(* CODESYS project Cat2.project

Project tree, tasks and I/O mapping:
  Device : CODESYS Control RTE V3, 3S - Smart Software Solutions GmbH, order no. 305017, version 3.5.11.0
    application Application
      libraries: Standard, * (System)
      task MainTask (cyclic, interval t#20ms, priority 1) calls PLC_PRG
      task VISU_TASK (cyclic, interval 100 ms, priority 31) calls VisuElems.Visu_Prg
      program PLC_PRG [ST]
      visualisation Visualization
      function block FB_Plant [ST]
      function block FB_Controller [ST]
      global variables GVL
      data type ST_PlantToController
      data type ST_ControllerToPlant
  text list GlobalTextList
  GlobalImagePool
*)

// Device/Application/ST_PlantToController
TYPE ST_PlantToController :
STRUCT
	// Buttons
	bCalibration : BOOL;
	bClean : BOOL;
	
	// Door
	bDoorOpened : BOOL;
	bDoorClosed : BOOL;
	
	// Separator
	bSeparatorUp : BOOL;
	bSeparatorDown : BOOL;
	
	// Weight
	CurrentWeight : REAL;
	
	// Wastes
	CurrentWastes : REAL;
	
	// Aroma
	CurrentAroma : REAL;

END_STRUCT
END_TYPE

// Device/Application/ST_ControllerToPlant
TYPE ST_ControllerToPlant :
STRUCT
	// Calibration
	bCalibration : BOOL;

	// Door
	bOpenDoor : BOOL;
	bCloseDoor : BOOL;
	bDoorStop : BOOL;
	
	// Separator
	bSeparatorUp : BOOL;
	bSeparatorDown : BOOL;
	
	// Aroma
	bAromaOn : BOOL;
	DeleteAroma : BOOL;
	
	// Wastes
	AddWastes : BOOL;
	
	// Weight
	FillerWeight : REAL;
	DeleteFiller : BOOL;
	
	bLowFiller : BOOL;
	bCriticalWastes : BOOL;
	bLowAroma : BOOL;
	AromaWorking : BOOL;
	
	UVworking : BOOL;
	
END_STRUCT
END_TYPE

// Device/Application/GVL

VAR_GLOBAL
	// Messages
	PlantToController : ST_PlantToController;
	ControllerToPlant : ST_ControllerToPlant;
	
	// Buttons
	CalibrationBtn : BOOL;
	CleanBtn : BOOL;
	
	AddCatBtn : BOOL;
	RemoveCatBtn : BOOL;
	
	RemoveWastesBtn : BOOL;
	RefillAromaBtn : BOOL;
	
	// Movements
	SeparatorPosition : REAL := 0.0;
	DoorPosition : REAL := 0.0;
	CatState : BOOL := FALSE;
	
	// Leds
	CalibrationLed : BOOL := FALSE;
	UVLed : BOOL;
	LowFillerLed : BOOL;
	FullWastesLed : BOOL;
	LowAromaLed : BOOL;
	AromaLed : BOOL;
	
	AddedFiller : REAL;
	CatWeight : REAL := 3.5;

END_VAR

// Device/Application/PLC_PRG
PROGRAM PLC_PRG
VAR
	Plant : FB_Plant;
	Controller : FB_Controller;
END_VAR

Plant();
Controller();

END_PROGRAM

// Device/Application/FB_Plant
FUNCTION_BLOCK FB_Plant
VAR_INPUT
END_VAR
VAR_OUTPUT
END_VAR

VAR CONSTANT
	FillerPart : REAL := 0.2;
	WastesPart : REAL := 5.0;
	AromaPart : REAL := 0.2;
	
	DoorMin : REAL := 0.0;
	DoorMax : REAL := 100.0;
	
	SeparatorMin : REAL := 270.0;
	SeparatorMax : REAL := 360.0;
END_VAR

VAR
	// Controller flags
	IsCalibration : BOOL := FALSE;
	IsCat : BOOL := FALSE;

	// Button triggers
	rtCalib : R_TRIG;
	CalibEvent : BOOL := FALSE;
	
	rtClean : R_TRIG;
	CleanEvent : BOOL := FALSE;
	
	rtAddCat : R_TRIG;
	rtRemoveCat : R_TRIG;
	
	rtRemoveWastes : R_TRIG;
	rtRefillAroma : R_TRIG;
	
	
	// Door movement
	DoorClose : BOOL := FALSE;
	DoorOpen : BOOL := FALSE;
	DoorOpening : BOOL := FALSE;
	DoorClosing : BOOL := FALSE;
	DoorClosed : BOOL := FALSE;
	DoorOpened : BOOL := FALSE;
	DoorPosition : REAL := DoorMin;
	
	// Separator movement
	SeparatorUp : BOOL := FALSE;
	flSepUp : F_TRIG;
	SeparatorDown : BOOL := FALSE;
	SeparatorUpping : BOOL := FALSE;
	SeparatorDowning : BOOL := FALSE;
	SeparatorUpped : BOOL := FALSE;
	SeparatorDowned : BOOL := FALSE;
	SeparatorPosition : REAL := SeparatorMax;
	
	// Weight
	CurrentWeight : REAL := 0.0;
	FillerWeight : REAL := 0.0;
	DeleteFiller : BOOL := FALSE;
	LowFiller : BOOL := FALSE;
	
	// Wastes
	CurrentWastesLevel : REAL := 0.0;
	AddWastes : BOOL := FALSE;
	CriticalWastes : BOOL := FALSE;
	
	// Aroma
	CurrentAromaLevel : REAL := 100.0;
	DeleteAroma : BOOL := FALSE;
	LowAroma : BOOL := FALSE;
	AromaWorking : BOOL := FALSE;
	flAroma : F_TRIG;
	
	UVworking : BOOL := FALSE;

END_VAR

// ==================== From Controller =======================
IsCalibration := GVL.ControllerToPlant.bCalibration;

DoorClose := GVL.ControllerToPlant.bCloseDoor;
DoorOpen := GVL.ControllerToPlant.bOpenDoor;
SeparatorUp := GVL.ControllerToPlant.bSeparatorUp;
SeparatorDown := GVL.ControllerToPlant.bSeparatorDown;

FillerWeight := GVL.ControllerToPlant.FillerWeight;
DeleteFiller := GVL.ControllerToPlant.DeleteFiller;

AddWastes := GVL.ControllerToPlant.AddWastes;

DeleteAroma := GVL.ControllerToPlant.DeleteAroma;

LowFiller := GVL.ControllerToPlant.bLowFiller;
LowAroma := GVL.ControllerToPlant.bLowAroma;
CriticalWastes := GVL.ControllerToPlant.bCriticalWastes;

UVworking := GVL.ControllerToPlant.UVworking;
AromaWorking := GVL.ControllerToPlant.AromaWorking;

// ==================== Button Events =======================
rtCalib(CLK := GVL.CalibrationBtn);
CalibEvent := rtCalib.Q;

rtAddCat(CLK := GVL.AddCatBtn);
rtRemoveCat(CLK := GVL.RemoveCatBtn);
IF rtAddCat.Q AND DoorOpened AND NOT IsCalibration THEN
	IsCat := TRUE;
ELSIF rtRemoveCat.Q AND DoorOpened THEN
	IsCat := FALSE;
END_IF

rtClean(CLK := GVL.CleanBtn);
CleanEvent := rtClean.Q;

rtRemoveWastes(CLK := GVL.RemoveWastesBtn);
rtRefillAroma(CLK := GVL.RefillAromaBtn);

IF rtRemoveWastes.Q AND NOT (SeparatorUpping OR SeparatorDowning) THEN
	CurrentWastesLevel := 0.0;
END_IF

IF rtRefillAroma.Q AND NOT AromaWorking THEN
	CurrentAromaLevel := 100.0;
END_IF

// ==================== Main =======================

// Calibration
IF IsCalibration THEN
	CurrentWeight := GVL.AddedFiller;
ELSIF IsCat THEN
	CurrentWeight := FillerWeight + GVL.CatWeight;
ELSE
	CurrentWeight := FillerWeight;
END_IF

// Door moving
IF DoorClose THEN
	DoorClosing := TRUE;
	DoorOpening := FALSE;
END_IF
	
IF DoorOpen THEN
	DoorClosing := FALSE;
	DoorOpening := TRUE;
END_IF

IF DoorOpen AND DoorClose THEN
	DoorClosing := FALSE;
	DoorOpening := FALSE;
END_IF

IF DoorClosing AND DoorPosition < DoorMax THEN
	DoorPosition := DoorPosition + 1;
	DoorClosed := FALSE;
	DoorOpened := FALSE;
ELSIF DoorOpening AND DoorPosition > DoorMin THEN
	DoorPosition := DoorPosition - 1;
	DoorClosed := FALSE;
	DoorOpened := FALSE;
END_IF

IF DoorPosition >= DoorMax THEN
	DoorPosition := DoorMax;
	DoorClosed := TRUE;
	DoorOpened := FALSE;
ELSIF DoorPosition <= DoorMin THEN
	DoorPosition := DoorMin;
	DoorOpened := TRUE;
	DoorClosed := FALSE;
END_IF

// Separator moving
flSepUp(CLK := SeparatorUp);

IF flSepUp.Q THEN
	IF (100 - CurrentWastesLevel) >= WastesPart THEN
		CurrentWastesLevel := CurrentWastesLevel + WastesPart;
	END_IF
	
	IF FillerWeight >= FillerPart THEN
		FillerWeight := FillerWeight - FillerPart;
		CurrentWeight := FillerWeight;
	END_IF
END_IF

IF SeparatorUp THEN
	SeparatorUpping := TRUE;
	SeparatorDowning := FALSE;
END_IF

IF SeparatorDown THEN
	SeparatorUpping := FALSE;
	SeparatorDowning := TRUE;
END_IF

IF SeparatorUp AND SeparatorDown THEN
	SeparatorUpping := FALSE;
	SeparatorDowning := FALSE;
END_IF

IF SeparatorUpping AND SeparatorPosition > SeparatorMin THEN
	SeparatorPosition := SeparatorPosition - 1;
	SeparatorUpped := FALSE;
	SeparatorDowned := FALSE;
ELSE
	SeparatorUpping := FALSE;
END_IF

IF SeparatorDowning AND SeparatorPosition < SeparatorMax THEN
	SeparatorPosition := SeparatorPosition + 1;
	SeparatorUpped := FALSE;
	SeparatorDowned := FALSE;
ELSE
	SeparatorDowning := FALSE;
END_IF

IF SeparatorPosition <= SeparatorMin THEN
	SeparatorPosition := SeparatorMin;
	SeparatorUpped := TRUE;
	SeparatorDowned := FALSE;
ELSIF SeparatorPosition >= SeparatorMax THEN
	SeparatorPosition := SeparatorMax;
	SeparatorUpped := FALSE;
	SeparatorDowned := TRUE;
END_IF

flAroma(CLK := AromaWorking);
IF flAroma.Q THEN
	IF CurrentAromaLevel >= AromaPart THEN
		CurrentAromaLevel := CurrentAromaLevel - AromaPart;
	END_IF
END_IF

// ==================== Positions =======================
GVL.DoorPosition := DoorPosition;
GVL.SeparatorPosition := SeparatorPosition;

// ==================== Leds =======================
GVL.CalibrationLed := IsCalibration;

GVL.CatState := IsCat;

GVL.FullWastesLed := CriticalWastes;
GVL.LowFillerLed := LowFiller;
GVL.LowAromaLed := LowAroma;

GVL.UVLed := UVworking;
GVL.AromaLed := AromaWorking;

// ==================== To Controller =======================
GVL.PlantToController.bCalibration := CalibEvent;
GVL.PlantToController.bClean := CleanEvent;

GVL.PlantToController.bDoorClosed := DoorClosed;
GVL.PlantToController.bDoorOpened := DoorOpened;
GVL.PlantToController.bSeparatorUp := SeparatorUpped;
GVL.PlantToController.bSeparatorDown := SeparatorDowned;

GVL.PlantToController.CurrentWeight := CurrentWeight;

GVL.PlantToController.CurrentWastes := CurrentWastesLevel;

GVL.PlantToController.CurrentAroma := CurrentAromaLevel;

END_FUNCTION_BLOCK

// Device/Application/FB_Controller
FUNCTION_BLOCK FB_Controller
VAR_INPUT
END_VAR
VAR_OUTPUT
END_VAR

VAR CONSTANT
	// Delay
	CatDelay : TIME := T#3S;
	SeparatorDelay : TIME := T#1S;
	UVdelay : TIME := T#4S;
	AromaDelay : TIME := T#2S;
	
	// Weight
	WeightTolerance : REAL := 0.02;
	LowFillerLevel : REAL := 0.5;
	LowAromaLevel : REAL := 0.05;
	CriticalWastesLevel : REAL := 90.0;
	
	VisitsToClean : INT := 5;
	
END_VAR

VAR
	LastState : INT := 0;
	CleaningState : INT := 0;
	State : INT := 0;
	
	VisitsCount : INT := 0;
	
	// Events
	CalibEvent : BOOL := FALSE;
	CleanEvent : BOOL := FALSE;
	
	// Flags
	CalibNow : BOOL := FALSE;
	
	CatNow : BOOL := FALSE;
	CatLeaved : BOOL := FALSE;
	CatDelayTimer : TON;
	
	CleaningNow : BOOL := FALSE;
	DoorMovingNow : BOOL := FALSE;
	
	UVnow : BOOL := FALSE;
	UVtimer : TON;
	
	AromaNow : BOOL := FALSE;
	
	// Door
	DoorClosed : BOOL := FALSE;
	DoorOpened : BOOL := FALSE;
	DoorOpening : BOOL := FALSE;
	DoorClosing : BOOL := FALSE;
	
	// Separator
	SeparatorUp : BOOL := FALSE;
	SeparatorDown : BOOL := FALSE;
	SeparatorUpping : BOOL := FALSE;
	SeparatorDowning : BOOL := FALSE;
	SeparatorDelayTimer : TON;
	SeparatorInDelay : BOOL := FALSE;
	
	// Weight
	CurrentWeight : REAL := 0;
	FillerWeight : REAL := 0;
	LowFiller : BOOL := FALSE;
	DeleteFiller : BOOL := FALSE;
	
	// Aroma
	CurrentAroma : REAL := 100.0;
	DeleteAroma : BOOL := FALSE;
	AromaTimer : TON;
	CriticalAroma : BOOL := FALSE;
	
	// Wastes
	CurrentWastes : REAL := 0.0;
	AddWastes : BOOL := FALSE;
	CriticalWastes : BOOL := FALSE;
	
END_VAR

CalibEvent := GVL.PlantToController.bCalibration;
CleanEvent := GVL.PlantToController.bClean;

DoorClosed := GVL.PlantToController.bDoorClosed;
DoorOpened := GVL.PlantToController.bDoorOpened;
SeparatorUp := GVL.PlantToController.bSeparatorUp;
SeparatorDown := GVL.PlantToController.bSeparatorDown;

CurrentWeight := GVL.PlantToController.CurrentWeight;
CurrentAroma := GVL.PlantToController.CurrentAroma;
CurrentWastes := GVL.PlantToController.CurrentWastes;

// Timers
CatDelayTimer(IN := CatLeaved, PT := SeparatorDelay);
SeparatorDelayTimer(IN := SeparatorInDelay, PT := SeparatorDelay);
UVtimer(IN := UVnow, PT := AromaDelay);
AromaTimer(IN := AromaNow, PT := AromaDelay);

DeleteFiller := FALSE;
AddWastes := FALSE;
DeleteAroma := FALSE;

IF DoorClosed AND State <> 1 THEN
	FillerWeight := CurrentWeight;
END_IF


CASE State OF
	0: // Zero state
		// Calibration event
		IF CalibEvent THEN
			LastState := 0;
			State := 10;
			RETURN;
		END_IF
		
		// Low aroma level
		IF CurrentAroma <= LowAromaLevel THEN
			CriticalAroma := TRUE;
		ELSE
			CriticalAroma := FALSE;
		END_IF
		
		// Critical wastes
		IF CurrentWastes >= CriticalWastesLevel THEN
			CriticalWastes := TRUE;
			State := 2;
			RETURN;
		ELSE
			CriticalWastes := FALSE;
		END_IF
		
		// Low filler
		IF FillerWeight <= LowFillerLevel THEN 
			LowFiller := TRUE;
			State := 1;
			RETURN;
		ELSE
			LowFiller := FALSE;
		END_IF
		
		// Cat in the litter box
		IF ABS(CurrentWeight - FillerWeight) > WeightTolerance THEN
			LastState := 0;
			State := 20;
			RETURN;
		ELSE
			FillerWeight := CurrentWeight;
		END_IF
		
		// Clean
		IF CleanEvent THEN
			LastState := 0;
			State := 40;
			RETURN;
		END_IF
		
	1: // Low filler level
		IF CalibEvent THEN
			State := 10;
		END_IF
		
	2: // Full wastes box
		IF CurrentWastes < CriticalWastesLevel THEN
			CriticalWastes := FALSE;
			State := 0;
		END_IF
		
	10: // Calibration
		CalibNow := TRUE;
		FillerWeight := CurrentWeight;
		IF CalibEvent THEN
			CalibNow := FALSE;
			State := 0;
		END_IF;
		
	20: // Cat here
		IF ABS(CurrentWeight - FillerWeight) <= WeightTolerance THEN
			CatLeaved := TRUE;
			VisitsCount := VisitsCount + 1;
			State := State + 1;
		END_IF
	
	21:
		IF ABS(CurrentWeight - FillerWeight) > WeightTolerance THEN
			CatLeaved := FALSE;
			State := State - 1;
		ELSIF CatDelayTimer.Q THEN
			CatLeaved := FALSE;
			State := State + 1;
		END_IF
	
	22:
		LastState := 22;
		State := 30;
		
	30: // Clening loop
		CASE LastState OF
			22: // Closing door
				State := 90;
			90: // Upping separator
				State := 100;
			100:
				SeparatorInDelay := TRUE;
				State := 102;
			102: // Downing separator
				SeparatorInDelay := FALSE;
				State := 101;
			101: // Opening door
				DeleteFiller := TRUE;
				AddWastes := TRUE;
				IF VisitsCount >= VisitsToClean THEN
					State := 40;
				ELSE
					State := 91;
				END_IF
			40:
				State := 91;
			91: // Finish
				State := 0;
				
		END_CASE
		LastState := 30;
	
	40: // UV and aroma
		CASE LastState OF
			0:
				CleaningState := 0;
				State := 90;
			30:
				UVnow := TRUE;
				CleaningState := 30;
				State := 110;
			90:
				UVnow := TRUE;
				State := 110;
			91:
				State := 0;
			110:
				UVnow := FALSE;
				AromaNow := NOT CriticalAroma;
				State := 120;
			120:
				VisitsCount := 0;
				AromaNow := FALSE;
				DeleteAroma := TRUE;
				IF CleaningState = 0 THEN
					State := 91;
				ELSE
					State := CleaningState;	
				END_IF			
		END_CASE
		LastState := 40;
		
	90: // Closing door
		DoorClosing := TRUE;
		IF DoorClosed THEN
			DoorClosing := FALSE;
			State := LastState;
			LastState := 90;
		END_IF
	
	91: // Opening door
		DoorOpening := TRUE;
		IF DoorOpened THEN
			DoorOpening := FALSE;
			State := LastState;
			LastState := 91;
		END_IF
		
	100: // Separator upping
		SeparatorUpping := TRUE;
		IF SeparatorUp THEN
			SeparatorUpping := FALSE;
			State := LastState;
			LastState := 100;
		END_IF
		
	101: // Separator downing
		SeparatorDowning := TRUE;
		IF SeparatorDown THEN
			SeparatorDowning := FALSE;
			State := LastState;
			LastState := 101;
		END_IF
	
	102: // Separator weiting
		IF SeparatorDelayTimer.Q THEN
			State := LastState;
			LastState := 102;
		END_IF
		
	110: // UV Cleaning
		IF UVtimer.Q THEN
			State := LastState;
			LastState := 110;
		END_IF
		
	120: // Aroma Working
		IF AromaTImer.Q OR CriticalAroma THEN
			State := LastState;
			LastState := 120;
		END_IF
END_CASE

GVL.ControllerToPlant.bCalibration := CalibNow;

GVL.ControllerToPlant.bCloseDoor := DoorClosing;
GVL.ControllerToPlant.bOpenDoor := DoorOpening;
GVL.ControllerToPlant.bSeparatorUp := SeparatorUpping;
GVL.ControllerToPlant.bSeparatorDown := SeparatorDowning;

GVL.ControllerToPlant.UVworking := UVnow;
GVL.ControllerToPlant.AromaWorking := AromaNow;

GVL.ControllerToPlant.FillerWeight := FillerWeight;
GVL.ControllerToPlant.DeleteFiller := DeleteFiller;

GVL.ControllerToPlant.AddWastes := AddWastes;
GVL.ControllerToPlant.DeleteAroma := DeleteAroma;

GVL.ControllerToPlant.bLowAroma := CriticalAroma;
GVL.ControllerToPlant.bLowFiller := LowFiller;
GVL.ControllerToPlant.bCriticalWastes := CriticalWastes;

END_FUNCTION_BLOCK

// Device/Application/Visualization
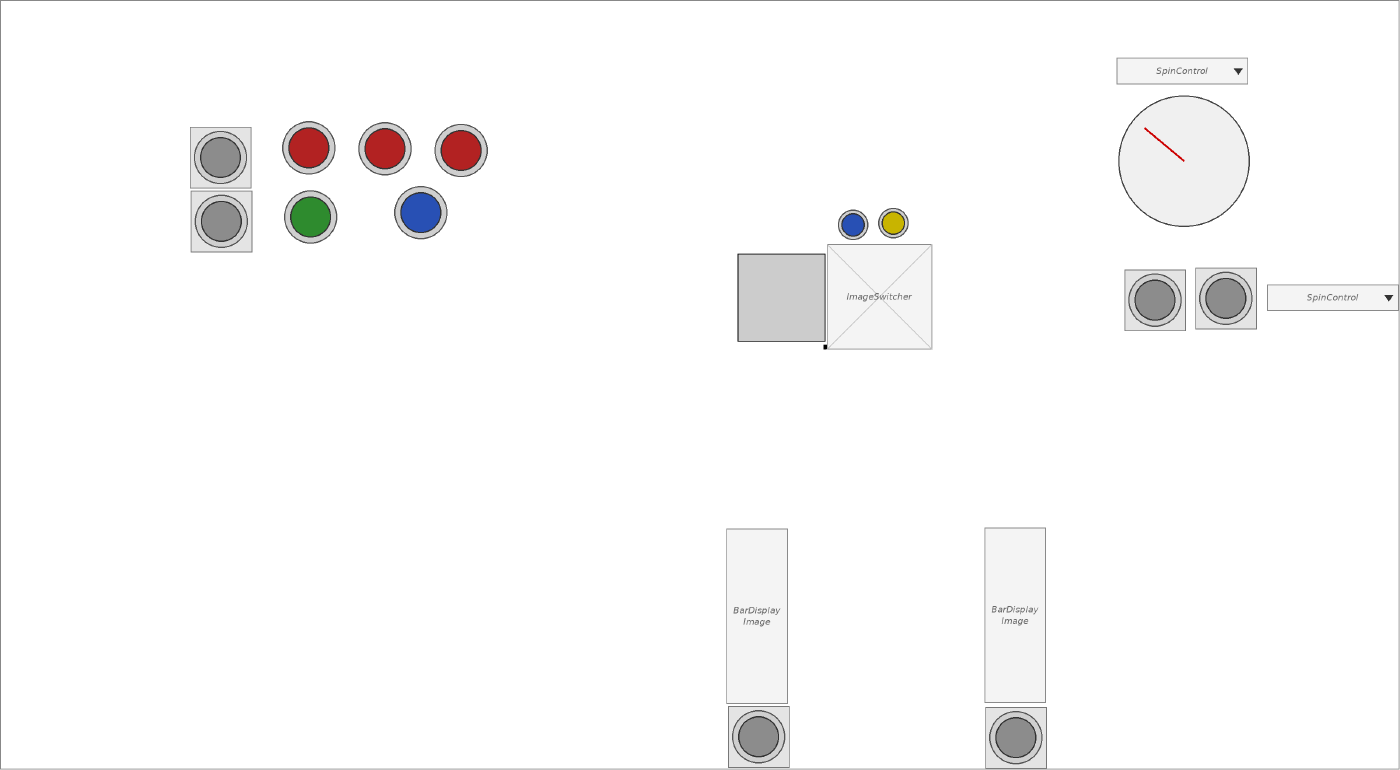
VISUALIZATION Visualization  // 1600x880
    PushSwitch (217,145 70x70), variable: CleanBtn, behaviour: TOGGLE, style: Switch-PushSwitch-Gray
    Rectangle (941,394 100x5)
        p2858320360: SeparatorPosition
    RoundedRectangle (843,290 100x100)
        p3560616238: DoorPosition
    ImageSwitcher (945,279 120x120), variable: CatState, background image: cat, behaviour: TOGGLE
    PushSwitch (218,218 70x70), variable: CalibrationBtn, behaviour: TOGGLE, style: Switch-PushSwitch-Gray
    PushSwitch (1285,308 70x70), variable: RemoveCatBtn, behaviour: TOGGLE, style: Switch-PushSwitch-Gray
    PushSwitch (1366,306 70x70), variable: AddCatBtn, behaviour: TOGGLE, style: Switch-PushSwitch-Gray
    PushSwitch (1126,808 70x70), variable: RefillAromaBtn, behaviour: TOGGLE, style: Switch-PushSwitch-Gray
    PushSwitch (832,807 70x70), variable: RemoveWastesBtn, behaviour: TOGGLE, style: Switch-PushSwitch-Gray
    BarDisplayImage (1125,603 70x200), value: PlantToController.CurrentAroma, style: BarDisplayImage-Gray, scale format: %.1f, scale 0..100
    BarDisplayImage (830,604 70x200), value: PlantToController.CurrentWastes, style: BarDisplayImage-Gray, scale format: %.1f, scale 0..100
    SpinControl (1448,325 150x30), variable: CatWeight
        p1653691745: 0.5
    Meter360 (1278,109 150x150), value: PlantToController.CurrentWeight, style: Meter-Meter360-Gray, scale format: %.1f, scale 0..20
    SpinControl (1276,66 150x30), variable: AddedFiller
        p1653691745: 0.5
    Lamp1 (320,213 70x70), variable: CalibrationLed, style: Lamp-Lamp1-Green
    Lamp1 (318,134 70x70), variable: LowFillerLed, style: Lamp-Lamp1-Red
    Lamp1 (405,135 70x70), variable: FullWastesLed, style: Lamp-Lamp1-Red
    Lamp1 (492,137 70x70), variable: LowAromaLed, style: Lamp-Lamp1-Red
    Lamp1 (446,208 70x70), variable: UVLed, style: Lamp-Lamp1-Blue
    Lamp1 (955,237 40x40), variable: UVLed, style: Lamp-Lamp1-Blue
    Lamp1 (1001,235 40x40), variable: AromaLed, style: Lamp-Lamp1-Yellow
END_VISUALIZATION
